PROGRAM MAIN
VAR
END_VAR

END_PROGRAM

(* stored: Version 1.1.0.1
   POU MAIN: Id {948ec821-0c9a-427d-b898-7036a31ff69a} *)
